// TwinCAT 3 PLC project Untitled1
// ProgramVersion: 3.1.4023.0
// libraries:
//   Tc2_Standard, * (Beckhoff Automation GmbH)
//   Tc2_System, * (Beckhoff Automation GmbH)
//   Tc3_Module, * (Beckhoff Automation GmbH)
// project tree:
//   / PlcTask.TcTTO
//   POUs/ MAIN.TcPOU
// real-time tasks:
//   TASK PlcTask: cycle T#10ms, priority 20, ADS port 350

CONFIGURATION Untitled1
    RESOURCE PLC ON TwinCAT3
        TASK PlcTask(INTERVAL := T#10ms, PRIORITY := 20);
        PROGRAM MAIN WITH PlcTask : MAIN;
    END_RESOURCE
END_CONFIGURATION

// ---- POUs/MAIN.TcPOU
PROGRAM MAIN
VAR
    RandomDintValue		: LREAL;
	fbDRAND				: DRAND;
	
	start				: BOOL;
	timer1				: TON;
END_VAR

timer1(IN := start, PT := T#1S,);

start := TRUE;
IF timer1.Q THEN
	fbDRAND(Seed := 1);
	
	RandomDintValue := 100*fbDRAND.Num;
	start := FALSE;
END_IF;

END_PROGRAM
